# EPICS StreamDevice protocol: templates/phase_add_support_submodule/support/@{device_support_module_name}/master/@{device_support_module_name}Sup/@{device_protocol_name}.proto
getIDN {
    out "*IDN?";
    in "%\$1[^\r\n]";
    ExtraInput = Ignore;
}

cmd {
    out "\$$1";
}

setD {
    out "\$1 %d";
}
getD {
    out "\$1?";
    in "%d";
    ExtraInput = Ignore;
}
